// TIA Portal V18 export
FUNCTION "IO MAP" : Void   // FC1, LAD
{ S7_Optimized_Access := 'FALSE' }
VERSION : 0.1
// stored: AutoNumber true, IsIECCheckEnabled false, SetENOAutomatically false, UDAEnableTagReadback false
BEGIN

REGION Network 1
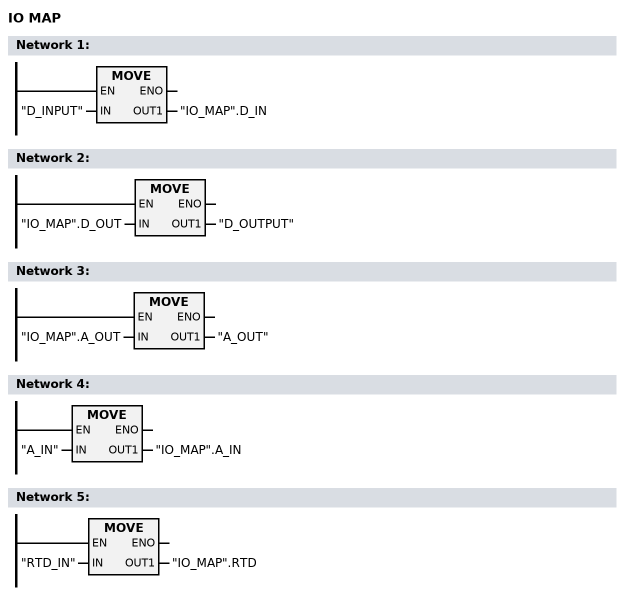
   RUNG wire#powerrail
      Move(in := "D_INPUT", out1 => "IO_MAP".D_IN)
   END_RUNG
   // the same network as SCL:
   "IO_MAP".D_IN := "D_INPUT";
END_REGION

REGION Network 2
   RUNG wire#powerrail
      Move(in := "IO_MAP".D_OUT, out1 => "D_OUTPUT")
   END_RUNG
   // the same network as SCL:
   "D_OUTPUT" := "IO_MAP".D_OUT;
END_REGION

REGION Network 3
   RUNG wire#powerrail
      Move(in := "IO_MAP".A_OUT, out1 => "A_OUT")
   END_RUNG
   // the same network as SCL:
   "A_OUT" := "IO_MAP".A_OUT;
END_REGION

REGION Network 4
   RUNG wire#powerrail
      Move(in := "A_IN", out1 => "IO_MAP".A_IN)
   END_RUNG
   // the same network as SCL:
   "IO_MAP".A_IN := "A_IN";
END_REGION

REGION Network 5
   RUNG wire#powerrail
      Move(in := "RTD_IN", out1 => "IO_MAP".RTD)
   END_RUNG
   // the same network as SCL:
   "IO_MAP".RTD := "RTD_IN";
END_REGION
END_FUNCTION
